VAR_GLOBAL RETAIN

END_VAR

(* stored: Version 1.1.0.1, ProductVersion 3.1.4022.7
   GVL Setup_Data: Id {e638b284-c167-45d9-89f1-3b43b5f206cc} *)
